TYPE ST_ExtController_get :
STRUCT
	control							: ST_ControlVars;
	Operation						: ST_OperationVars;
	SoftSettings					: ST_SoftSettings;
	HardSettings					: ST_HardSettings;
	events							: ST_ExtController_Events;
	b_AdvancedControl				: BOOL;
	ui_Heartbeat					: UINT;
	s_dashboardID					: STRING;
	b_Active						: BOOL;
	e_ConnectionState				: eConnectionState;
	s_OutputJson					: STRING(2000);
	LoggingBudgetOK					: BOOL := TRUE;
END_STRUCT
END_TYPE

(* stored: Version 1.1.0.1, ProductVersion 3.1.4026.18
   DUT ST_ExtController_get: Id {d5515538-88f2-47fe-9ec6-cb1b22314c01} *)
